// TIA Portal V21 export
TYPE "Std_EthFlowMeter"
   STRUCT
      Volume_flow : Real;   // Portata volumetrica (m³/h)
      Mass_Flow : Real;   // Portata massica (kg/h)
      Corrected_Volume_Flow : Real;   // Portata volumetrica (kg/h)
      Velocity : Real;
      Totalizer_1 : Real;   // m³
      Totalizer_2 : Real;   // l
      Totalizer_3 : Real;   // l
      ControlTotalizzatore_1 : Byte;   // 0=Avvia 1=Reset+Mantieni 2=PreimpostatoMantieni 3=Azzera+Totalizza 4=Preimpostato+Tot 5=HoldMantieni
      ControlTotalizzatore_2 : Byte;   // 0=Avvia 1=Reset+Mantieni 2=PreimpostatoMantieni 3=Azzera+Totalizza 4=Preimpostato+Tot 5=HoldMantieni
      ControlTotalizzatore_3 : Byte;   // 0=Avvia 1=Reset+Mantieni 2=PreimpostatoMantieni 3=Azzera+Totalizza 4=Preimpostato+Tot 5=HoldMantieni
   END_STRUCT;
END_TYPE
